Staubli VAL3: onStart.pgx

program onStart()
  local num i
  local num l_nClock
  local num l_nResult
  local string l_sSession
  local string l_sMessage
  local string l_sEmpty
begin
  // logMsg
  logMsg("[KERNEL] INTERFACE:PAGE Select program")
  // BUILD THE LIST
  l_sEmpty=""
  sProgType="PROG"
  nProgID=0
  // disable the filter
  if saveData:mode<2
    saveData:sProgFilter=""
  endIf
  // load the progType
  call load()
  // define the list
  call buildList()
  // record the old value....
  call use:selectNewField(nSelected,nIndex,nView)
  // build the page
  use:bUseRefresh=true
  //
end
